(* PLC project Lib2dMath, Beckhoff Automation GmbH TwinCAT PLC Control 3.5.13.21 *)
(* stored: creationDateTime 2024-03-30T11:42:44.2492878, modificationDateTime 2024-03-30T11:42:44.2492878 *)

TYPE udtVector : UNION
  v : udtVectorData;
  Koordinate : ARRAY[0..1] OF LREAL;
END_UNION;
END_TYPE
